FUNCTION_BLOCK FB_Btn
VAR_INPUT
	xStart:BOOL;
	xStop:BOOL;
	xReset:BOOL;
	xNextPas:BOOL;
	xAru:BOOL;
	xAirPressureOk : BOOL;
	iMotorSpeed: INT;
	
	//Auto mode
	xAllowedGetPiece: BOOL;
	xPiecePresent : BOOL;
	xEmulateZDone : BOOL;
	
	//Init Mode
	xHomingPosReached : BOOL;
	xJogXForward : BOOL;
	xJogXBackward: BOOL;
	xJogYForward : BOOL;
	xJogYBackward: BOOL;
	
	//Btn used in Manual-Mode
	xSetHomePos : BOOL;
	xManualAct1GoIn: BOOL;
	xManualAct1GoOut : BOOL;
END_VAR

END_FUNCTION_BLOCK

(* stored: Version 1.1.0.1, ProductVersion 3.1.4020.12
   POU FB_Btn: Id {9d1b347e-0701-4dd1-a9e2-079105cb34be}, SpecialFunc None *)
